SUBAPPLICATION Ventilsteuerung_Uebung_100 (* DigitalInput_I1 auf DigitalOutput_Q1, mit Plug and Socket *)
  (* Standard: 61499-2 *)
  (* Version 1.0, 2023-10-23, franz *)
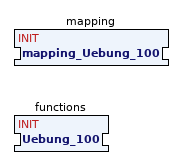
  SUBAPPS
    mapping : mapping_Uebung_100;
    functions : Uebung_100;
  END_SUBAPPS
END_SUBAPPLICATION
